FUNCTION_BLOCK TWO_I_TWO_O (* Extracted Composite Function Block Type *)
  (* Standard: 61499-2 *)
  (* Version 9/9/2026, lizar *)
  PACKAGE Main;
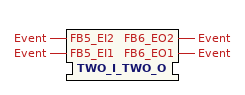
  EVENT_INPUT
    FB5_EI2; (* Second input event *)
    FB5_EI1; (* First input event *)
  END_EVENT
  EVENT_OUTPUT
    FB6_EO2; (* Second output event,etc. *)
    FB6_EO1; (* First output event *)
  END_EVENT
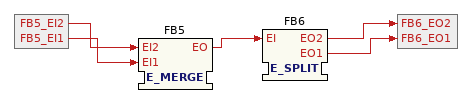
  FBS
    FB5 : E_MERGE;
    FB6 : E_SPLIT;
  END_FBS
  EVENT_CONNECTIONS
    FB5.EO TO FB6.EI;
    FB5_EI2 TO FB5.EI2;
    FB5_EI1 TO FB5.EI1;
    FB6.EO2 TO FB6_EO2;
    FB6.EO1 TO FB6_EO1;
  END_CONNECTIONS
END_FUNCTION_BLOCK
